(* CODESYS project LD_Function.pou_xml.xml

Project tree, tasks and I/O mapping:
  function LD_Function [LD]
*)

// LD_Function
FUNCTION LD_Function : BOOL
VAR_INPUT
	xStart : BOOL;
	xStop_NC : BOOL;
END_VAR
VAR_OUTPUT
	xPump : BOOL;
END_VAR

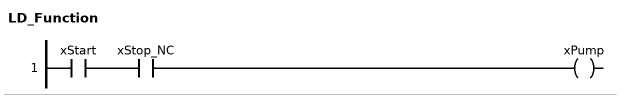
// NETWORK 1
xPump := xStart AND xStop_NC;

END_FUNCTION
